// TIA Portal V20 export
TYPE "UDT_OPC_ActualValuesAxis"
   STRUCT
      StationNumber : Byte;
      AxisId : DInt;
      ActualPosition : LReal;
   END_STRUCT;
END_TYPE
